{attribute 'qualified_only'}
{attribute 'strict'}
TYPE E_ModbusState :
(
	enum_member := 0
);
END_TYPE

(* stored: Version 1.1.0.1, ProductVersion 3.1.4020.14
   DUT E_ModbusState: Id {3df81ecc-0810-4a27-8334-ebc9859a7779} *)
